(* PLC project cab, Dassault Systèmes ControlBuild 2024x *)
(* stored: creationDateTime 2023-10-03T11:13:51-01:00 *)

PROGRAM tni_train.cab
  VAR_INPUT
    keyCabEnabled2 : BOOL := false;
    keyCabDisabled2 : BOOL := false;
  END_VAR
  VAR_OUTPUT
    enableOpeningRightC1 : BOOL := false;
    enableOpeningLeftC1 : BOOL := false;
    enableClosingRightC1 : BOOL := false;
    enableClosingLeftC1 : BOOL := false;
  END_VAR
  VAR_OUTPUT
    cabEnabled : BOOL := false;
    cabDisabled : BOOL := false;
    cabIncoherence : BOOL := false;
  END_VAR

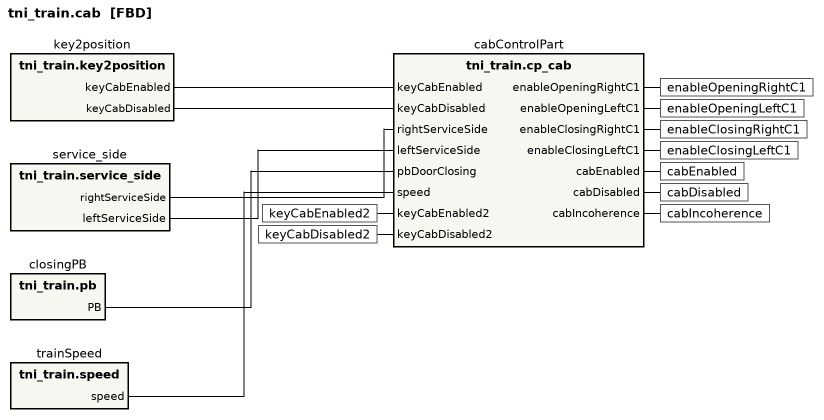
(* FBD diagram, written out as Structured Text *)
key2position();
service_side();
closingPB();
trainSpeed();
cabControlPart(keyCabEnabled := key2position.keyCabEnabled, keyCabDisabled := key2position.keyCabDisabled, rightServiceSide := service_side.rightServiceSide, leftServiceSide := service_side.leftServiceSide, pbDoorClosing := closingPB.PB, speed := trainSpeed.speed, keyCabEnabled2 := keyCabEnabled2, keyCabDisabled2 := keyCabDisabled2);
enableOpeningRightC1 := cabControlPart.enableOpeningRightC1;
enableOpeningLeftC1 := cabControlPart.enableOpeningLeftC1;
enableClosingRightC1 := cabControlPart.enableClosingRightC1;
enableClosingLeftC1 := cabControlPart.enableClosingLeftC1;
cabEnabled := cabControlPart.cabEnabled;
cabDisabled := cabControlPart.cabDisabled;
cabIncoherence := cabControlPart.cabIncoherence;
END_PROGRAM
